{attribute 'qualified_only'}
{attribute 'strict'}
TYPE E_BoxHookPoint :
(
	
	Origin 		:= 0,
	Station_1	:= 1,
	Station_2	:= 2,
	Station_3	:= 3,
	Station_4	:= 4,
	Station_5	:= 5,
	Station_6	:= 6,
	Station_7	:= 7,
	Station_8	:= 8,
	Station_9	:= 9,
	
);
END_TYPE

(* stored: Version 1.1.0.1, ProductVersion 3.1.4024.13
   DUT E_BoxHookPoint: Id {cb65c850-c959-4442-afec-60079a2ed718} *)
